{attribute 'hide_all_locals'}
{attribute 'conditionalshow'}
FUNCTION_BLOCK FB_PID
VAR_INPUT
	{attribute 'hide'}
	bEnable					: BOOL;						//Enable the regulation
	{attribute 'hide'}
	rSetpoint				: REAL;						//Setpoint to which the controller controls
	{attribute 'hide'}
	udiIValue				: UDINT;					//Reset time
	{attribute 'hide'}
	udiDValue				: UDINT;					//Lead time
	{attribute 'hide'}
	udiDamping				: UDINT;					//Damping
	{attribute 'hide'}
	rPValue					: REAL;						//Controller gain
	{attribute 'hide'}
	rMaxValue				: REAL;						//Max Value from the output of the controller
	{attribute 'hide'}
	rMinValue				: REAL;						//Min Value from the output of the controller
	{attribute 'hide'}
	rNeutralZone			: REAL;						//If the value of the control deviation is smaller than half of lrNeutralZone, the control signal remains the same
	{attribute 'hide'}
	bDirection				: BOOL;						//Direction from the controller
	{attribute 'hide'}
	rActualValue			: REAL;						//Current value that the controller tries to adapt to the setpoint and to regulate
END_VAR
VAR_OUTPUT
	{attribute 'hide'}
	rQController			: REAL;						//Controller output
END_VAR
VAR
	PIDController			: FB_BA_PIDCtrl;			//PID controller
END_VAR

//Creator : Kai Ebensperger
//Company : Lynus AG
//Date : 19.05.2021
//Version : 1.0.0.0

//This function block represents a classic PID controller that can be set individually.
PIDController(
	bEn:= bEnable, 
	rW:= rSetpoint, 
	rX:= rActualValue, 
	udiOpMode:= 0, 
	bActn:= bDirection, 
	rKp:= rPValue, 
	udiTn_ms:= udiIValue, 
	udiTv_ms:= udiDValue, 
	udiTd_ms:= udiDamping, 
	rYMax:= rMaxValue, 
	rYMin:= rMinValue, 
	rNZ:= rNeutralZone, 
	udiCycCl:= 1, 
	bSync:= , 
	rSync:= , 
	rY=> rQController, 
	rE=> , 
	bARW=> );

END_FUNCTION_BLOCK

(* stored: Version 1.1.0.1, ProductVersion 3.1.4024.6
   POU FB_PID: Id {4bfdfe12-8044-48cc-b265-f47876182ca5}, SpecialFunc None *)
